// TIA Portal V17 export
// export: Created 2025-04-11T04:54:22.7154014Z, ExportSetting WithDefaults, DisplayName Totally Integrated Automation Portal, DisplayVersion V17, DisplayName TIA Portal Openness, DisplayVersion V17, DisplayName TIA Portal Version Control Interface, DisplayVersion V17, DisplayName SINAMICS Startdrive Advanced, DisplayVersion V17, DisplayName SINAMICS Startdrive G130, G150, S120, S150, SINAMICS MV, S210, DisplayVersion V17, DisplayName SINAMICS Startdrive G110M, G120, G120C, G120D, G120P, G115D, DisplayVersion V17, DisplayName STEP 7 Professional, DisplayVersion V17, DisplayName STEP 7 Safety, DisplayVersion V17, DisplayName WinCC Advanced, DisplayVersion V17
VAR_GLOBAL   // PLC tag table "默认变量表"
END_VAR
VAR_GLOBAL CONSTANT   // user constants
   "1#氢气探测器" : Int := 0;
   "2#氢气探测器" : Int := 1;
   "1#火焰探测器" : Int := 2;
   "2#火焰探测器" : Int := 3;
   "1#主电机电流反馈" : Int := 4;
   "2#主电机电流反馈" : Int := 5;
   "备用(37)" : Int := 6;
   "备用(38)" : Int := 7;
   仪表风压力 : Int := 8;
   进气压力 : Int := 9;
   一级排气压力 : Int := 10;
   二级排气压力 : Int := 11;
   隔离腔压力1 : Int := 12;
   隔离腔压力2 : Int := 13;
   液压油压力1 : Int := 14;
   液压油压力2 : Int := 15;
   进气冷却前温度 : Int := 16;
   进气冷却后温度 : Int := 17;
   一级排气冷却前温度 : Int := 18;
   一级排气冷却后温度 : Int := 19;
   二级排气冷却前温度 : Int := 20;
   二级排气冷却后温度 : Int := 21;
   冷却水入口温度 : Int := 22;
   冷却水出口温度 : Int := 23;
   液压油温度 : Int := 24;   // 55
   液压油液位 : Int := 25;
   缸1转子流量计 : Int := 26;
   缸2转子流量计 : Int := 27;
   "备用(16)" : Int := 28;
   "备用(22)" : Int := 29;
   "备用(23)" : Int := 30;
   "备用(24)" : Int := 31;
END_VAR
